// TIA Portal V16 export
// export: Created 2022-06-10T08:04:28.5128801Z, ExportSetting WithDefaults, DisplayName Totally Integrated Automation Portal, DisplayVersion V16, DisplayName TIA Portal Version Control Interface, DisplayVersion V16, DisplayName TIA Portal Openness, DisplayVersion V16, DisplayName TIA Portal Teamcenter Gateway, DisplayVersion V16, DisplayName STEP 7 Professional, DisplayVersion V16, DisplayName SINUMERIK ONE STEP 7 Toolbox, DisplayVersion V16, DisplayName STEP 7 Safety, DisplayVersion V16, DisplayName SINUMERIK 840D sl STEP 7 Toolbox, DisplayVersion V16, DisplayName WinCC Advanced, DisplayVersion V16
FUNCTION "Absaugung" : Void   // FC302, STL
TITLE = Absauganlage
{ S7_Optimized_Access := 'FALSE' }
AUTHOR : TBE_STO
FAMILY : 5S4517
NAME : JGWS
VERSION : 0.1
// stored: AutoNumber false, ParameterPassing false, UDAEnableTagReadback false
   VAR_TEMP
      inputVorwarnug : Bool;
      inputVerschmutzt : Bool;
      timeVorwarnung : Bool;
      timeVerschmutzt : Bool;
      timeKarrenz : Bool;
      timeRest : DInt;
   END_VAR
BEGIN

NETWORK
TITLE = Absauganlage: vorhanden ???
// Quelle 5g  => Absauganlage
      AN    "Allgemein".absaug_vorh;
      BEC;


NETWORK
TITLE = Absauganlage: Motorschutzschalter
      AN    "absMotorschutz_e";
      S     "LBP_AlarmMsgs".UserA[13].A70UUxx[1];


NETWORK
TITLE = Absauganlage: Sammelstörung
      A     "NULL";
      A     "absaug_ti_aktiv";
      S     "LBP_AlarmMsgs".UserA[13].A70UUxx[5];


NETWORK
TITLE = Absauganlage: Betriebsbereit fehlt
      AN    "EINS";
      A     "absaug_ti_aktiv";
      S     "LBP_AlarmMsgs".UserA[13].A70UUxx[6];


NETWORK
TITLE = Filterüberwachung Versorgung Eingang Vorwarnung
      A(;
      O     "IOL_IN81";
      O     "IOL_IN82";
      );
      A     "Allgemein".absaug_filter_IOL;
      O;
      A(;
      ON    "absBereit_e";
      ON    "EINS";
      );
      AN    "Allgemein".absaug_filter_IOL;
      =     #inputVorwarnug;

NETWORK
TITLE = Filterüberwachung Versorgung Eingang Verschmutzt
      A     "IOL_IN81";
      A     "Allgemein".absaug_filter_IOL;
      O;
      AN    "absBereit_e";
      AN    "Allgemein".absaug_filter_IOL;
      =     #inputVerschmutzt;

NETWORK
TITLE = Sollzeitüberwachung: Minimalwert 600 Sekunden
      L     "Allgemein".absaug_filter_time_soll;
      L     600;
      >=D;
      JC    FSOL;
      T     "Allgemein".absaug_filter_time_soll;
FSOL: NOP   0;


NETWORK
TITLE = Karrenzzeit berechnen, Standard 8 Stunden
      L     "Allgemein".absaug_filter_time_soll;
      L     29100;
      <=D;
      L     300;
      JC    RST0;
      L     "Allgemein".absaug_filter_time_soll;
      L     28800;
      -D;
RST0: T     #timeRest;


NETWORK
TITLE = Filterüberwachung Vorwarnung
      A(;
      L     "Allgemein".absaug_filter_time_ist;
      L     60;
      >=D;
      );
      =     #timeVorwarnung;


NETWORK
TITLE = Filterüberwachung Verschmutzt
      A(;
      L     "Allgemein".absaug_filter_time_ist;
      L     "Allgemein".absaug_filter_time_soll;
      >=D;
      );
      =     #timeVerschmutzt;


NETWORK
TITLE = Filterüberwachung Karrenzzeit Verschmutzt
      A(;
      L     "Allgemein".absaug_filter_time_ist;
      L     #timeRest;
      >D;
      );
      =     #timeKarrenz;


NETWORK
TITLE = Filterüberwachung Zeitzähler
      AN    "absaug_ti_aktiv";
      ON    "takt1sZyklus";
      JC    FEND;

      AN    #inputVorwarnug;
      AN    #inputVerschmutzt;
      O     #timeVerschmutzt;
      JC    FRUK;
      L     "Allgemein".absaug_filter_time_ist;
      +     DINT#1;
      T     "Allgemein".absaug_filter_time_ist;
      JU    FEND;

FRUK: L     "Allgemein".absaug_filter_time_ist;
      L     0;
      <=D;
      O     #inputVorwarnug;
      O     #inputVerschmutzt;
      JC    FEND;
      L     "Allgemein".absaug_filter_time_ist;
      +     DINT#-1;
      T     "Allgemein".absaug_filter_time_ist;

FEND: NOP   0;


NETWORK
TITLE = Absauganlage: Filter ist verschmutzt Vorwarnung
// U     DB2.DBX  290.7
//       L     S5T#10M
//       SE    T    273
      A     #inputVorwarnug;
      A     #timeVorwarnung;
      A     "Allgemein".absaug_filter;
      A     "absaug_ti_aktiv";
      S     "LBP_AlarmMsgs".UserA[13].A70UUxx[55];
      A     "LBP_AlarmMsgs".UserA[13].A70UUxx[7];
      R     "LBP_AlarmMsgs".UserA[13].A70UUxx[55];
      A     "LBP_AlarmMsgs".UserA[13].A70UUxx[55];
      S     "lampeOrangeBlink";


NETWORK
TITLE = Absauganlage: Filter ist verschmutzt
      A     #inputVerschmutzt;
      A     #timeVerschmutzt;
      A     "Allgemein".absaug_filter;
      A     "absaug_ti_aktiv";
      S     "LBP_AlarmMsgs".UserA[13].A70UUxx[7];


NETWORK
TITLE = Absauganlage: Filter ist verschmutzt Karrenzzeit
      A     #timeKarrenz;
      A     "Allgemein".absaug_filter;
      =     "LBP_AlarmMsgs".UserA[13].A70UUxx[54];


NETWORK
TITLE = Karrenzzeit durch Einrichrter nachtriggern
      AN    "eks_einrichter";
      ON    "msttStörungLöschen";
      ON    #timeKarrenz;
      JC    TKAR;
      L     #timeRest;
      L     200;
      -D;
      T     "Allgemein".absaug_filter_time_ist;
TKAR: NOP   0;


NETWORK
TITLE = Absauganlage: Strömungsüberwachung 1 Vorwarnung
      A(;
      AN    "IOL_IN84";
      A     "Allgemein".absaug_stroem_IOL;
      O;
      A     "EINS";
      AN    "Allgemein".absaug_stroem_IOL;
      );
      A     "Allgemein".absaug_stroem;
      A     "uf_sp_geschl";
      A     "absaug_ti_aktiv";
      AN    "absaug_ti_stroem1";
      =     "LBP_AlarmMsgs".UserA[13].A70UUxx[52];
      A     "LBP_AlarmMsgs".UserA[13].A70UUxx[52];
      S     "lampeOrangeBlink";


NETWORK
TITLE = Absauganlage: Strömungsüberwachung 1
      A(;
      AN    "IOL_IN83";
      A     "Allgemein".absaug_stroem_IOL;
      O;
      A     "NULL";
      AN    "Allgemein".absaug_stroem_IOL;
      );
      A     "Allgemein".absaug_stroem;
      A     "uf_sp_geschl";
      A     "absaug_ti_aktiv";
      L     S5T#10S;
      SD    "absaug_ti_stroem1";
      NOP   0;
      NOP   0;
      NOP   0;
      A     "absaug_ti_stroem1";
      S     "LBP_AlarmMsgs".UserA[13].A70UUxx[15];


NETWORK
TITLE = Absauganlage: Strömungsüberwachung 2 Vorwarnung
      A(;
      AN    "EINS";
      A     "Allgemein".absaug_stroem_IOL;
      O;
      A     "NULL";
      AN    "Allgemein".absaug_stroem_IOL;
      );
      A     "Allgemein".absaug_stroem;
      A     "uf_sp_geschl";
      A     "absaug_ti_aktiv";
      AN    "absaug_ti_stroem2";
      =     "LBP_AlarmMsgs".UserA[13].A70UUxx[53];
      A     "LBP_AlarmMsgs".UserA[13].A70UUxx[53];
      S     "lampeOrangeBlink";


NETWORK
TITLE = Absauganlage: Strömungsüberwachung 2
      A(;
      AN    "EINS";
      A     "Allgemein".absaug_stroem_IOL;
      O;
      A     "NULL";
      AN    "Allgemein".absaug_stroem_IOL;
      );
      A     "Allgemein".absaug_stroem;
      A     "uf_sp_geschl";
      A     "absaug_ti_aktiv";
      L     S5T#10S;
      SD    "absaug_ti_stroem2";
      NOP   0;
      NOP   0;
      NOP   0;
      A     "absaug_ti_stroem2";
      S     "LBP_AlarmMsgs".UserA[13].A70UUxx[23];


NETWORK
TITLE = Absauganlage: Motor einschalten
      A(;
      O     "kn1ProgLaeuft";
      O     "kn2ProgLaeuft";
      O     "kn3ProgLaeuft";
      O     "kn4ProgLaeuft";
      );
      L     "Allgemein".absaug_nachlauf;
      SF    "absaug_ti_ein";


NETWORK
TITLE = Absauganlage: Reaktion
      O     "LBP_AlarmMsgs".UserA[13].A70UUxx[1];
      O     "LBP_AlarmMsgs".UserA[13].A70UUxx[5];
      O     "LBP_AlarmMsgs".UserA[13].A70UUxx[6];
      ON    "notHaltOk_m";
      R     "absaug_ti_ein";


NETWORK
TITLE = Absauganlage: Motor einschalten
      A     "absaug_ti_ein";
      AN    "GreenPlus".einh_4_Standby_aktiv;
      A     "ma_aktiv_energie";
      =     "absEin_a";


NETWORK
TITLE = Absauganlage: Meldung Not-Halt
      A     "notHaltOk";
      =     "allg_ausgeng";
//Relais Maschine kein Not-Halt


NETWORK
TITLE = Absauganlage: Motor ist aktiv
      A     "absaug_ti_ein";
      AN    "GreenPlus".einh_4_Standby_aktiv;
      A     "ma_aktiv_energie";
      L     S5T#5S;
      SD    "absaug_ti_aktiv";


NETWORK
TITLE = Absauganlage: Reaktion
      O     "LBP_AlarmMsgs".UserA[13].A70UUxx[1];
      O     "LBP_AlarmMsgs".UserA[13].A70UUxx[5];
      O     "LBP_AlarmMsgs".UserA[13].A70UUxx[6];
      O     "LBP_AlarmMsgs".UserA[13].A70UUxx[7];
      O     "LBP_AlarmMsgs".UserA[13].A70UUxx[15];
      O     "LBP_AlarmMsgs".UserA[13].A70UUxx[23];
      S     "nck <<_ss KN";


NETWORK
TITLE = Baustein Ende
      BEU;


NETWORK
TITLE = Absauganlage deaktiviert
ENDE: A     "EINS";
      R     "absEin_a";


NETWORK
TITLE = Absauganlage deaktiviert
      L     0;
      T     "Allgemein".absaug_filter_time_ist;

END_FUNCTION
